// SIMATIC S7-200 project (STEP 7-Micro/WIN), CPU 224XP REL 02.01

SYMBOL_TABLE USUARIO1
P_MARCHA         I0.0
FC_2_ABAJO       I0.1
FC_3_ARRIBA      I0.2
FC_4_IZQUIERDA   I0.3
FC_5_DERECHA     I0.4
SUBIR            Q0.0
BAJAR            Q0.1
DERECHA          Q0.2
IZQUIERDA        Q0.3
CONTROL          MB1
END_SYMBOL_TABLE

ORGANIZATION_BLOCK PRINCIPAL:OB1
TITLE=COMENTARIOS DEL PROGRAMA
BEGIN
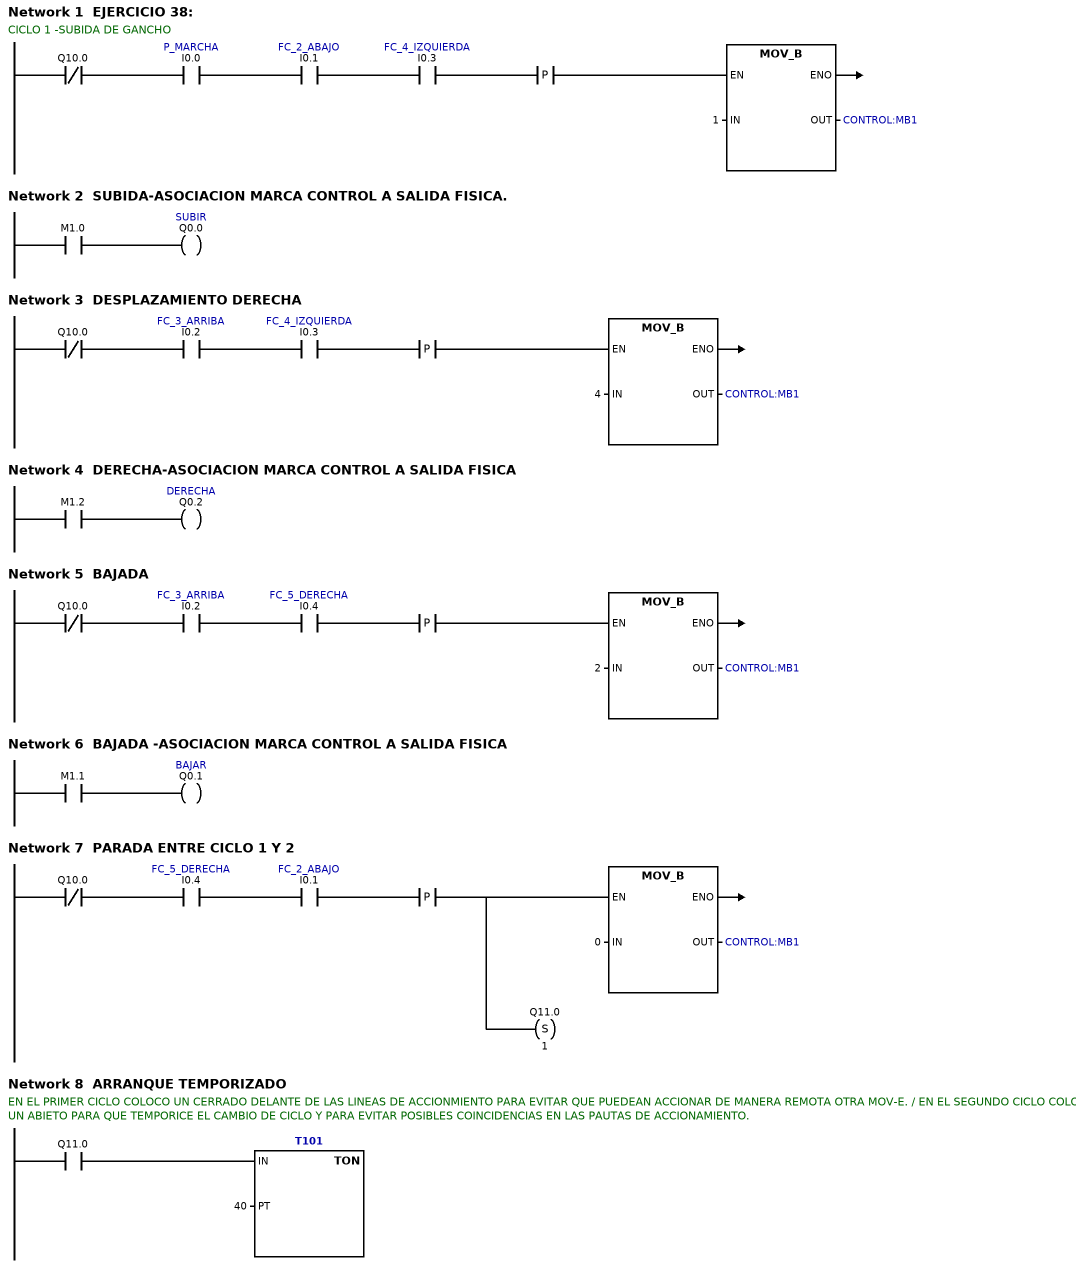
Network 1 // EJERCICIO 38:
// CICLO 1 -SUBIDA DE GANCHO
LDN    Q10.0
A      P_MARCHA:I0.0
A      FC_2_ABAJO:I0.1
A      FC_4_IZQUIERDA:I0.3
EU
MOVB   1, CONTROL:MB1
Network 2 // SUBIDA-ASOCIACION MARCA CONTROL A SALIDA FISICA.
LD     M1.0
=      SUBIR:Q0.0
Network 3 // DESPLAZAMIENTO DERECHA
LDN    Q10.0
A      FC_3_ARRIBA:I0.2
A      FC_4_IZQUIERDA:I0.3
EU
MOVB   4, CONTROL:MB1
Network 4 // DERECHA-ASOCIACION MARCA CONTROL A SALIDA FISICA
LD     M1.2
=      DERECHA:Q0.2
Network 5 // BAJADA
LDN    Q10.0
A      FC_3_ARRIBA:I0.2
A      FC_5_DERECHA:I0.4
EU
MOVB   2, CONTROL:MB1
Network 6 // BAJADA -ASOCIACION MARCA CONTROL A SALIDA FISICA
LD     M1.1
=      BAJAR:Q0.1
Network 7 // PARADA ENTRE CICLO 1 Y 2 
LDN    Q10.0
A      FC_5_DERECHA:I0.4
A      FC_2_ABAJO:I0.1
EU
MOVB   0, CONTROL:MB1
S      Q11.0, 1
Network 8 // ARRANQUE TEMPORIZADO
// EN EL PRIMER CICLO COLOCO UN CERRADO DELANTE DE LAS LINEAS DE ACCIONMIENTO PARA EVITAR QUE PUEDEAN ACCIONAR DE MANERA REMOTA OTRA MOV-E.
// EN EL SEGUNDO CICLO COLOCO UN ABIETO PARA QUE TEMPORICE EL CAMBIO DE CICLO Y PARA EVITAR POSIBLES COINCIDENCIAS EN LAS PAUTAS DE ACCIONAMIENTO.
LD     Q11.0
TON    T101, 40
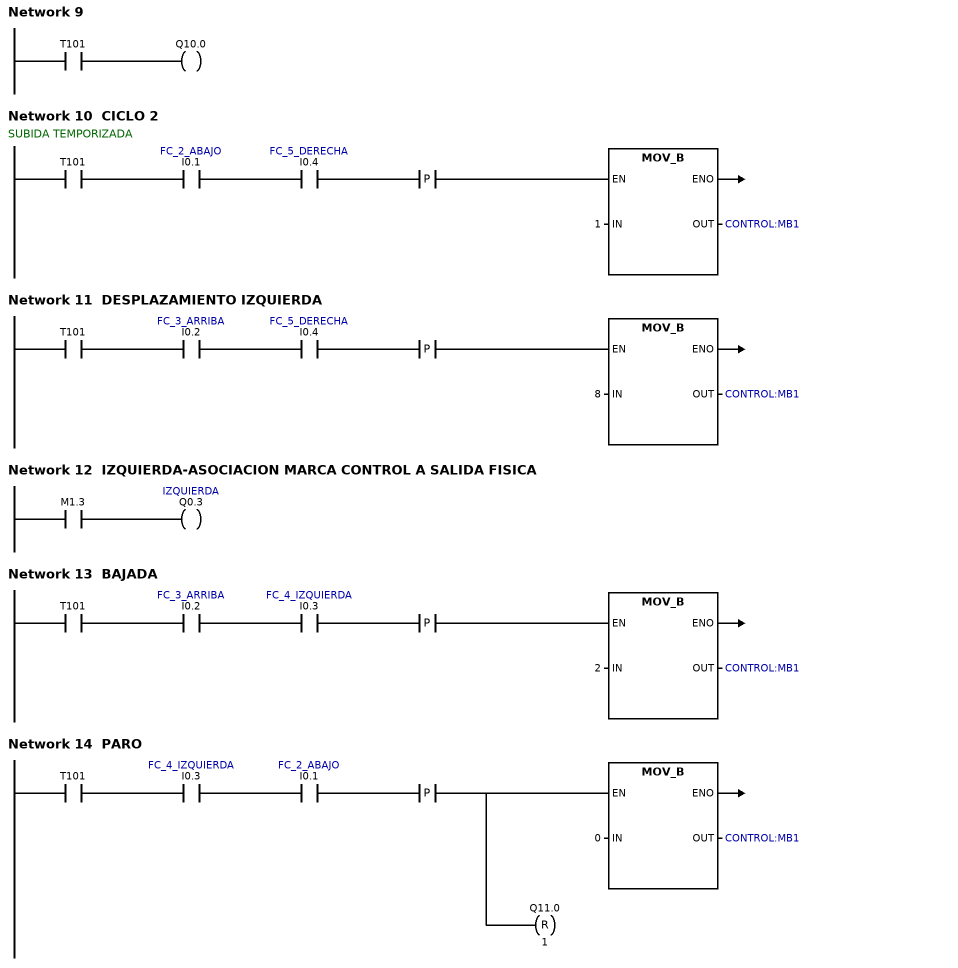
Network 9
LD     T101
=      Q10.0
Network 10 // CICLO 2 
// SUBIDA TEMPORIZADA
// (network saved uncompiled; LAD cells follow)
// row 0: c0 -| |- T101  c1 -| |- FC_2_ABAJO:I0.1  c2 -| |- FC_5_DERECHA:I0.4  c3 -|P|-  c4 --  c5 [MOV_B EN:=power@row0, IN:=1, ENO=>power, OUT=>CONTROL:MB1]  c6 ->
// row 1: c5 [box]
Network 11 // DESPLAZAMIENTO IZQUIERDA
// (network saved uncompiled; LAD cells follow)
// row 0: c0 -| |- T101  c1 -| |- FC_3_ARRIBA:I0.2  c2 -| |- FC_5_DERECHA:I0.4  c3 -|P|-  c4 --  c5 [MOV_B EN:=power@row0, IN:=8, ENO=>power, OUT=>CONTROL:MB1]  c6 ->
// row 1: c5 [box]
Network 12 // IZQUIERDA-ASOCIACION MARCA CONTROL A SALIDA FISICA
LD     M1.3
=      IZQUIERDA:Q0.3
Network 13 // BAJADA
// (network saved uncompiled; LAD cells follow)
// row 0: c0 -| |- T101  c1 -| |- FC_3_ARRIBA:I0.2  c2 -| |- FC_4_IZQUIERDA:I0.3  c3 -|P|-  c4 --  c5 [MOV_B EN:=power@row0, IN:=2, ENO=>power, OUT=>CONTROL:MB1]  c6 ->
// row 1: c5 [box]
Network 14 // PARO
// (network saved uncompiled; LAD cells follow)
// row 0: c0 -| |- T101  c1 -| |- FC_4_IZQUIERDA:I0.3  c2 -| |- FC_2_ABAJO:I0.1  c3 -|P|-  v  c4 --  c5 [MOV_B EN:=power@row0, IN:=0, ENO=>power, OUT=>CONTROL:MB1]  c6 ->
// row 1: c3 ^v  c5 [box]
// row 2: c3 ^  c4 -(R) Q11.0, 1
END_ORGANIZATION_BLOCK
